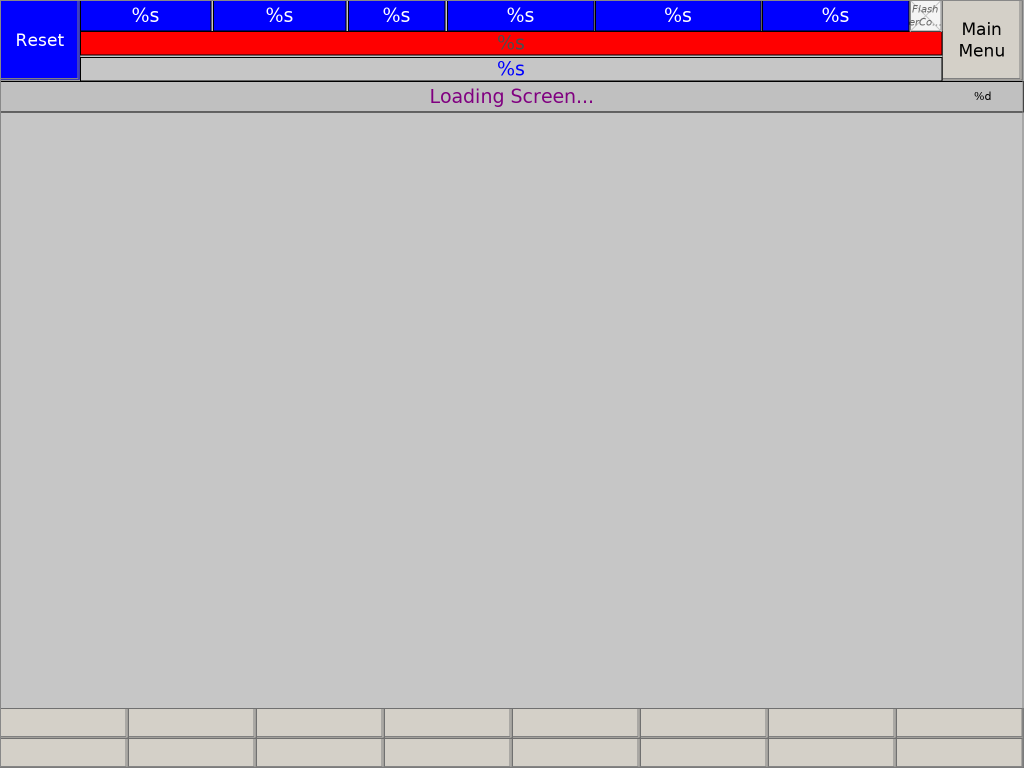
VISUALIZATION Tmp_001_Template_Alternate  // 1024x768
VAR_IN_OUT
	header:typeHMIheader;
	
END_VAR
    Rectangle (595,0 166x31)
        p2167032090: header.AnyStationWarningColour
    Rectangle (80,57 862x24)
    Group (0,0 1022x80)
        Button (0,0 80x80), "Reset"
            tap gHMIButtons.btnReset
            OnMouseDown: execute { gHMIButtons.gAnyButtonPressed := TRUE; }
        Button (942,0 80x80), "Main Menu"
            OnMouseClick: change screen: Men_030_MenuScreen
            OnMouseDown: execute { gHMIButtons.gAnyButtonPressed := TRUE; }
    Group (80,31 862x24)
        Rectangle (0,0 862x24), "%s", text variable: GlobalMessages.gMsgMc.Warning.topMessage, invisible if: gHMIData.gHideDisplayElementWarningView.McEnabled
        Rectangle (0,0 862x24), "%s", text variable: GlobalMessages.gMsgS1.Warning.topMessage, invisible if: gHMIData.gHideDisplayElementWarningView.S1Enabled
        Rectangle (0,0 862x24), "%s", text variable: GlobalMessages.gMsgS2.Warning.topMessage, invisible if: gHMIData.gHideDisplayElementWarningView.S2Enabled
        Rectangle (0,0 862x24), "%s", text variable: GlobalMessages.gMsgS3.Warning.topMessage, invisible if: gHMIData.gHideDisplayElementWarningView.S3Enabled
        Rectangle (0,0 862x24), "%s", text variable: GlobalMessages.gMsgS4.Warning.topMessage, invisible if: gHMIData.gHideDisplayElementWarningView.S4Enabled
        Rectangle (0,0 862x24), "%s", text variable: GlobalMessages.gMsgS5.Warning.topMessage, invisible if: gHMIData.gHideDisplayElementWarningView.S5Enabled
        Rectangle (0,0 862x24), "%s", text variable: GlobalMessages.gMsgS6.Warning.topMessage, invisible if: gHMIData.gHideDisplayElementWarningView.S6Enabled
    Group (80,31 862x24)
        OnMouseClick: change screen: Msg_020_Alarms
        Rectangle (0,0 862x24), "%s", text variable: GlobalMessages.gMsgMc.Alarm.topMessage, invisible if: gHMIData.gHideDisplayElementAlarmView.McEnabled
        Rectangle (0,0 862x24), "%s", text variable: GlobalMessages.gMsgS1.Alarm.topMessage, invisible if: gHMIData.gHideDisplayElementAlarmView.S1Enabled, text list: ''
        Rectangle (0,0 862x24), "%s", text variable: GlobalMessages.gMsgS2.Alarm.topMessage, invisible if: gHMIData.gHideDisplayElementAlarmView.S2Enabled
        Rectangle (0,0 862x24), "%s", text variable: GlobalMessages.gMsgS3.Alarm.topMessage, invisible if: gHMIData.gHideDisplayElementAlarmView.S3Enabled
        Rectangle (0,0 862x24), "%s", text variable: GlobalMessages.gMsgS4.Alarm.topMessage, invisible if: gHMIData.gHideDisplayElementAlarmView.S4Enabled
        Rectangle (0,0 862x24), "%s", text variable: GlobalMessages.gMsgS5.Alarm.topMessage, invisible if: gHMIData.gHideDisplayElementAlarmView.S5Enabled
        Rectangle (0,0 862x24), "%s", text variable: GlobalMessages.gMsgS6.Alarm.topMessage, invisible if: gHMIData.gHideDisplayElementAlarmView.S6Enabled
    Group (80,57 862x24)
        Rectangle (0,0 862x24), "%s", text variable: GlobalMessages.gMsgMc.Prompts.topMessage, invisible if: gHMIData.gHideDisplayElementPromptView.McEnabled
        Rectangle (0,0 862x24), "%s", text variable: GlobalMessages.gMsgS1.Prompts.topMessage, invisible if: gHMIData.gHideDisplayElementPromptView.S1Enabled
        Rectangle (0,0 862x24), "%s", text variable: GlobalMessages.gMsgS2.Prompts.topMessage, invisible if: gHMIData.gHideDisplayElementPromptView.S2Enabled
        Rectangle (0,0 862x24), "%s", text variable: GlobalMessages.gMsgS3.Prompts.topMessage, invisible if: gHMIData.gHideDisplayElementPromptView.S3Enabled
        Rectangle (0,0 862x24), "%s", text variable: GlobalMessages.gMsgS4.Prompts.topMessage, invisible if: gHMIData.gHideDisplayElementPromptView.S4Enabled
        Rectangle (0,0 862x24), "%s", text variable: GlobalMessages.gMsgS5.Prompts.topMessage, invisible if: gHMIData.gHideDisplayElementPromptView.S5Enabled
        Rectangle (0,0 862x24), "%s", text variable: GlobalMessages.gMsgS6.Prompts.topMessage, invisible if: gHMIData.gHideDisplayElementPromptView.S6Enabled
    Rectangle (0,81 1024x31), "Loading Screen...", text list: 'ScreenNames', text index: gHMIData.gScreenNumber
    Rectangle (595,0 166x31), "%s", colour toggle: header.AnyStationFaultHeaderActive, invisible if: NOT header.isAnyFaultState, text list: 'AnyStationAlarmList', text index: header.AnyStationFaultHeader
        p2167032090: header.AnyStationFaultColour
    Group (80,0 861x31)
        Rectangle (0,0 131x31), "%s", text list: 'ModeStatesHeader', text index: header.stationstate
        Rectangle (133,0 133x31), "%s", text list: 'CycleType', text index: header.cycleTypeFeedback
        Rectangle (268,0 97x31), "%s", colour toggle: header.isFaultState, text list: 'FaultState', text index: header.FaultStateHeader
        Rectangle (682,0 147x31), "%s", text list: 'StationNames', text index: header.stationNameSelect
            OnMouseClick: OpenDialog Dialog=dialogStation, OpenModal=True, PositionX=100, PositionY=250
        Rectangle (367,0 147x31), "%s", colour toggle: header.homestateColour, text list: 'HomeState', text index: header.homestate
        Image (830,0 31x31), invisible if: header.flasher, image: FlasherCorner.aus
        Image (830,0 31x31), invisible if: NOT header.flasher, image: FlasherCorner.ein
    Rectangle (595,0 166x31), "%s", colour toggle: header.AnyStationWarningHeaderActive, invisible if: NOT header.isAnyWarningState, text list: 'AnyStationWarningList', text index: header.AnyStationWarningHeader
        p2167032090: header.AnyStationWarningColour
    Rectangle (945,81 76x31), "%d", text variable: gHMIData.gScreenNumber
    Button (0,738 128x30)
        OnMouseDown: execute { gHMIButtons.gAnyButtonPressed := TRUE; }
    Button (128,738 128x30)
        OnMouseDown: execute { gHMIButtons.gAnyButtonPressed := TRUE; }
    Button (256,738 128x30)
        OnMouseDown: execute { gHMIButtons.gAnyButtonPressed := TRUE; }
    Button (384,738 128x30)
        OnMouseDown: execute { gHMIButtons.gAnyButtonPressed := TRUE; }
    Button (512,738 128x30)
        OnMouseDown: execute { gHMIButtons.gAnyButtonPressed := TRUE; }
    Button (640,738 128x30)
        OnMouseDown: execute { gHMIButtons.gAnyButtonPressed := TRUE; }
    Button (768,738 128x30)
        OnMouseDown: execute { gHMIButtons.gAnyButtonPressed := TRUE; }
    Button (896,738 128x30)
        OnMouseDown: execute { gHMIButtons.gAnyButtonPressed := TRUE; }
    Button (0,708 128x30)
        OnMouseDown: execute { gHMIButtons.gAnyButtonPressed := TRUE; }
    Button (128,708 128x30)
        OnMouseDown: execute { gHMIButtons.gAnyButtonPressed := TRUE; }
    Button (256,708 128x30)
        OnMouseDown: execute { gHMIButtons.gAnyButtonPressed := TRUE; }
    Button (384,708 128x30)
        OnMouseDown: execute { gHMIButtons.gAnyButtonPressed := TRUE; }
    Button (512,708 128x30)
        OnMouseDown: execute { gHMIButtons.gAnyButtonPressed := TRUE; }
    Button (640,708 128x30)
        OnMouseDown: execute { gHMIButtons.gAnyButtonPressed := TRUE; }
    Button (768,708 128x30)
        OnMouseDown: execute { gHMIButtons.gAnyButtonPressed := TRUE; }
    Button (896,708 128x30)
        OnMouseDown: execute { gHMIButtons.gAnyButtonPressed := TRUE; }
END_VISUALIZATION

(* stored: Version 1.1.0.1, ProductVersion 3.1.4024.11
   Visu Tmp_001_Template_Alternate: Id {96dc712c-0044-0203-0349-4d1fd957007b} *)
